// TIA Portal V19 export
VAR_GLOBAL   // PLC tag table "Em0"
   "Signal stack yellow" AT %Q34.1 : Bool;   // Yellow signal stack light
   "Signal stack horn" AT %Q34.4 : Bool;   // Horn on signal stack
   "Signal stack red" AT %Q34.0 : Bool;   // Red signal stack light
   "Signal stack green" AT %Q34.3 : Bool;   // Green signal stack light
   "Signal stack blue" AT %Q34.2 : Bool;   // Blue signal stack light
   "Signal stack white" AT %Q34.5 : Bool;   // White signal stack light
END_VAR
